(* IEC 61131-3 sources: AXOpen/src/components.drives/ctrl/src/AxoDrives (part 2) *)

            //*************AXO_MOVE_VELOCITY************
            _movementInPositiveDirection := _AxoMoveVelocity_Velocity > 0 AND _AxoMoveVelocity_Direction = AXOpen.Components.Abstractions.Drives.eAxoDriveDirection#PositiveDirection OR
                                            _AxoMoveVelocity_Velocity < 0 AND _AxoMoveVelocity_Direction = AXOpen.Components.Abstractions.Drives.eAxoDriveDirection#NegativeDirection;
            _movementInNegativeDirection := _AxoMoveVelocity_Velocity < 0 AND _AxoMoveVelocity_Direction = AXOpen.Components.Abstractions.Drives.eAxoDriveDirection#PositiveDirection OR
                                            _AxoMoveVelocity_Velocity > 0 AND _AxoMoveVelocity_Direction = AXOpen.Components.Abstractions.Drives.eAxoDriveDirection#NegativeDirection;
                                            AxoMoveVelocity_Task.SetIsDisabled(_movementDisabled OR (_movementInPositiveDirection AND NOT EnablePositive)  OR (_movementInNegativeDirection AND NOT EnableNegative) );
            THIS.MC_MoveVelocity(AxisRef,
                        AxoMoveVelocity_Task.Execute(THIS),
                        _AxoMoveVelocity_ContinuousUpdate,
                        _AxoMoveVelocity_Velocity,
                        _AxoMoveVelocity_Acceleration,
                        _AxoMoveVelocity_Deceleration,
                        _AxoMoveVelocity_Jerk,
                        _AxoMoveVelocity_Direction,
                        AxoMoveVelocity_InVelocity,
                        AxoMoveVelocity_Busy,
                        AxoMoveVelocity_Active,
                        AxoMoveVelocity_CommandAborted,
                        AxoMoveVelocity_Error,
                        AxoMoveVelocity_ErrorID);

            IF AxoMoveVelocity_Task.IsBusy() THEN
                IF AxoMoveVelocity_Task.IsFirstExecutionCycle() THEN
                    AxoMoveVelocity_ContinuousUpdate    :=  _AxoMoveVelocity_ContinuousUpdate;
                    AxoMoveVelocity_Velocity            :=  _AxoMoveVelocity_Velocity;
                    AxoMoveVelocity_Acceleration        :=  _AxoMoveVelocity_Acceleration;
                    AxoMoveVelocity_Deceleration        :=  _AxoMoveVelocity_Deceleration;
                    AxoMoveVelocity_Jerk                :=  _AxoMoveVelocity_Jerk;
                    AxoMoveVelocity_Direction           :=  _AxoMoveVelocity_Direction;
                END_IF;
                AxoMoveVelocity_Task.DoneWhen(AxoMoveVelocity_InVelocity AND NOT _AxoMoveVelocity_ContinuousUpdate);
                AxoMoveVelocity_Task.ThrowWhen(AxoMoveVelocity_Error,CONCAT('<#MC_MoveVelocity has thrown an error: #>', ToString(AxoMoveVelocity_ErrorID)));
                IF AxoMoveVelocity_CommandAborted THEN
                    AxoMoveVelocity_Task.Abort();
                END_IF;
            END_IF;
            IF AxoMoveVelocity_Task.RestoreTriggered() OR AxoMoveVelocity_Task.AbortTriggered() THEN;
                AxoMoveVelocity_InVelocity := FALSE;
            END_IF;
            //******************************************

            //*************AXO_TORQUE_CONTROL***********
            _movementInPositiveDirection := _AxoTorqueControl_Torque > 0 AND _AxoTorqueControl_Direction = AXOpen.Components.Abstractions.Drives.eAxoDriveDirection#PositiveDirection OR
                                            _AxoTorqueControl_Torque < 0 AND _AxoTorqueControl_Direction = AXOpen.Components.Abstractions.Drives.eAxoDriveDirection#NegativeDirection;
            _movementInNegativeDirection := _AxoTorqueControl_Torque < 0 AND _AxoTorqueControl_Direction = AXOpen.Components.Abstractions.Drives.eAxoDriveDirection#PositiveDirection OR
                                            _AxoTorqueControl_Torque > 0 AND _AxoTorqueControl_Direction = AXOpen.Components.Abstractions.Drives.eAxoDriveDirection#NegativeDirection;
            AxoTorqueControl_Task.SetIsDisabled(_movementDisabled OR (_movementInPositiveDirection AND NOT EnablePositive)  OR (_movementInNegativeDirection AND NOT EnableNegative) );
            THIS.MC_TorqueControl(AxisRef,
                        AxoTorqueControl_Task.Execute(THIS),
                        _AxoTorqueControl_ContinuousUpdate,
                        _AxoTorqueControl_Torque,
                        _AxoTorqueControl_TorqueRamp,
                        _AxoTorqueControl_PositionLimit,
                        _AxoTorqueControl_Velocity,
                        _AxoTorqueControl_Acceleration,
                        _AxoTorqueControl_Deceleration,
                        _AxoTorqueControl_Jerk,
                        _AxoTorqueControl_Direction,
                        AxoTorqueControl_InTorque,
                        AxoTorqueControl_Busy,
                        AxoTorqueControl_Active,
                        AxoTorqueControl_CommandAborted,
                        AxoTorqueControl_Error,
                        AxoTorqueControl_ErrorID);

            IF AxoTorqueControl_Task.IsBusy() THEN
                IF AxoTorqueControl_Task.IsFirstExecutionCycle() THEN
                    AxoTorqueControl_ContinuousUpdate   :=  _AxoTorqueControl_ContinuousUpdate;
                    AxoTorqueControl_Torque             :=  _AxoTorqueControl_Torque;
                    AxoTorqueControl_TorqueRamp         :=  _AxoTorqueControl_TorqueRamp;
                    AxoTorqueControl_PositionLimit      :=  _AxoTorqueControl_PositionLimit;
                    AxoTorqueControl_Velocity           :=  _AxoTorqueControl_Velocity;
                    AxoTorqueControl_Acceleration       :=  _AxoTorqueControl_Acceleration;
                    AxoTorqueControl_Deceleration       :=  _AxoTorqueControl_Deceleration;
                    AxoTorqueControl_Jerk               :=  _AxoTorqueControl_Jerk;
                    AxoTorqueControl_Direction          :=  _AxoTorqueControl_Direction;
                END_IF;
                AxoTorqueControl_Task.DoneWhen(AxoTorqueControl_InTorque AND NOT _AxoTorqueControl_ContinuousUpdate);
                AxoTorqueControl_Task.ThrowWhen(AxoTorqueControl_Error,CONCAT('<#MC_TorqueControl has thrown an error: #>', ToString(AxoTorqueControl_ErrorID)));
                IF AxoTorqueControl_CommandAborted THEN
                    AxoTorqueControl_Task.Abort();
                END_IF;
            END_IF;
            IF AxoTorqueControl_Task.RestoreTriggered() OR AxoTorqueControl_Task.AbortTriggered() THEN;
                AxoTorqueControl_InTorque := FALSE;
            END_IF;
            //******************************************
            IF DriveState = eAxoDriveState#ContinuousMotion AND (ActualVelocity > 0.5 AND NOT EnablePositive OR ActualVelocity < -0.5 AND NOT EnableNegative) THEN
                _disabledDuringMovement := TRUE;
                IF AxoMoveVelocity_Task.IsBusy() THEN
                    AxoMoveVelocity_Task.Restore();
                END_IF;
                IF AxoTorqueControl_Task.IsBusy() THEN
                    AxoTorqueControl_Task.Restore();
                END_IF;
            END_IF;
            //*************AXO_SET_POSITION*************
            AxoSetPosition_Task.SetIsDisabled(FALSE);
            THIS.MC_SetPosition(AxisRef,
                        AxoSetPosition_Task.Execute(THIS),
                        _AxoSetPosition_Position,
                        _AxoSetPosition_Relative,
                        _AxoSetPosition_ExecutionMode,
                        AxoSetPosition_Done,
                        AxoSetPosition_Busy,
                        AxoSetPosition_Error,
                        AxoSetPosition_ErrorID);

            IF AxoSetPosition_Task.IsBusy() THEN
                AxoSetPosition_Task.DoneWhen(AxoSetPosition_Done);
                AxoSetPosition_Task.ThrowWhen(AxoSetPosition_Error,CONCAT('<#MC_SetPosition has thrown an error: #>', ToString(AxoSetPosition_ErrorID)));
            END_IF;
            //******************************************

            //*************AXO_SET_OVERRIDE*************
            AxoSetOverride_Task.SetIsDisabled(FALSE);
            AxoSetOverride_Task.Run(THIS);
            THIS.MC_SetOverride(AxisRef,
                        AxoSetOverride_Task.IsSwitchedOn(),
                        _AxoSetOverride_VelFactor,
                        _AxoSetOverride_AccFactor,
                        _AxoSetOverride_JerkFactor,
                        AxoSetOverride_Enabled,
                        AxoSetOverride_Busy,
                        AxoSetOverride_Error,
                        AxoSetOverride_ErrorID);
            //******************************************

            //*************AXO_READ_PARAMETER***********
            AxoReadParameter_Task.SetIsDisabled(FALSE);
            AxoReadParameter_Task.Run(THIS);
            THIS.MC_ReadParameter(AxisRef,
                        AxoReadParameter_Task.IsSwitchedOn(),
                        _AxoReadParameter_ParameterNumber,
                        AxoReadParameter_Valid,
                        AxoReadParameter_Busy,
                        AxoReadParameter_Error,
                        AxoReadParameter_ErrorID,
                        AxoReadParameter_Value);
            IF  AxoReadParameter_Task.IsSwitchedOff() THEN
                AxoReadParameter_Valid := FALSE;
                AxoReadParameter_Value := LINT#0;
            END_IF;
            //******************************************

            //*************AXO_READ_REAL_PARAMETER******
            AxoReadRealParameter_Task.SetIsDisabled(FALSE);
            AxoReadRealParameter_Task.Run(THIS);
            THIS.MC_ReadRealParameter(AxisRef,
                        AxoReadRealParameter_Task.IsSwitchedOn(),
                        _AxoReadRealParameter_ParameterNumber,
                        AxoReadRealParameter_Valid,
                        AxoReadRealParameter_Busy,
                        AxoReadRealParameter_Error,
                        AxoReadRealParameter_ErrorID,
                        AxoReadRealParameter_Value);
            IF  AxoReadRealParameter_Task.IsSwitchedOff() THEN
                AxoReadRealParameter_Valid := FALSE;
                AxoReadRealParameter_Value := REAL#0.0;
            END_IF;
            //******************************************

            //*************AXO_READ_BOOL_PARAMETER******
            AxoReadBoolParameter_Task.SetIsDisabled(FALSE);
            AxoReadBoolParameter_Task.Run(THIS);
            THIS.MC_ReadBoolParameter(AxisRef,
                        AxoReadBoolParameter_Task.IsSwitchedOn(),
                        _AxoReadBoolParameter_ParameterNumber,
                        AxoReadBoolParameter_Valid,
                        AxoReadBoolParameter_Busy,
                        AxoReadBoolParameter_Error,
                        AxoReadBoolParameter_ErrorID,
                        AxoReadBoolParameter_Value);
            IF  AxoReadBoolParameter_Task.IsSwitchedOff() THEN
                AxoReadBoolParameter_Valid := FALSE;
                AxoReadBoolParameter_Value := FALSE;
            END_IF;
            //******************************************

            //*************AXO_WRITE_PARAMETER**********
            AxoWriteParameter_Task.SetIsDisabled(FALSE);
            THIS.MC_WriteParameter(AxisRef,
                        AxoWriteParameter_Task.Execute(THIS),
                        _AxoWriteParameter_ParameterNumber,
                        _AxoWriteParameter_Value,
                        _AxoWriteParameter_ExecutionMode,
                        AxoWriteParameter_Done,
                        AxoWriteParameter_Busy,
                        AxoWriteParameter_Error,
                        AxoWriteParameter_ErrorID);
            IF AxoWriteParameter_Task.IsBusy() THEN
                AxoWriteParameter_Task.DoneWhen(AxoWriteParameter_Done);
                AxoWriteParameter_Task.ThrowWhen(AxoWriteParameter_Error,CONCAT('<#MC_WriteParameter has thrown an error: #>', ToString(AxoWriteParameter_ErrorID)));
            END_IF;
            //******************************************

            //*************AXO_WRITE_REAL_PARAMETER*****
            AxoWriteRealParameter_Task.SetIsDisabled(FALSE);
            THIS.MC_WriteRealParameter(AxisRef,
                        AxoWriteRealParameter_Task.Execute(THIS),
                        _AxoWriteRealParameter_ParameterNumber,
                        _AxoWriteRealParameter_Value,
                        _AxoWriteRealParameter_ExecutionMode,
                        AxoWriteRealParameter_Done,
                        AxoWriteRealParameter_Busy,
                        AxoWriteRealParameter_Error,
                        AxoWriteRealParameter_ErrorID);
            IF AxoWriteRealParameter_Task.IsBusy() THEN
                AxoWriteRealParameter_Task.DoneWhen(AxoWriteRealParameter_Done);
                AxoWriteRealParameter_Task.ThrowWhen(AxoWriteRealParameter_Error,CONCAT('<#MC_WriteRealParameter has thrown an error: #>', ToString(AxoWriteRealParameter_ErrorID)));
            END_IF;
            //******************************************

            //*************AXO_WRITE_BOOL_PARAMETER*****
            AxoWriteBoolParameter_Task.SetIsDisabled(FALSE);
            THIS.MC_WriteBoolParameter(AxisRef,
                        AxoWriteBoolParameter_Task.Execute(THIS),
                        _AxoWriteBoolParameter_ParameterNumber,
                        _AxoWriteBoolParameter_Value,
                        _AxoWriteBoolParameter_ExecutionMode,
                        AxoWriteBoolParameter_Done,
                        AxoWriteBoolParameter_Busy,
                        AxoWriteBoolParameter_Error,
                        AxoWriteBoolParameter_ErrorID);
            IF AxoWriteBoolParameter_Task.IsBusy() THEN
                AxoWriteBoolParameter_Task.DoneWhen(AxoWriteBoolParameter_Done);
                AxoWriteBoolParameter_Task.ThrowWhen(AxoWriteBoolParameter_Error,CONCAT('<#MC_WriteBoolParameter has thrown an error: #>', ToString(AxoWriteBoolParameter_ErrorID)));
            END_IF;
            //******************************************

            //*************AXO_READ_DIGITAL_INPUT*******
            AxoReadDigitalInput_Task.SetIsDisabled(FALSE);
            AxoReadDigitalInput_Task.Run(THIS);
            THIS.MC_ReadDigitalInput(AxisRef,
                        AxoReadDigitalInput_Task.IsSwitchedOn(),
                        _AxoReadDigitalInput_InputNumber,
                        AxoReadDigitalInput_Valid,
                        AxoReadDigitalInput_Busy,
                        AxoReadDigitalInput_Error,
                        AxoReadDigitalInput_ErrorID,
                        AxoReadDigitalInput_Value);
            IF  AxoReadDigitalInput_Task.IsSwitchedOff() THEN
                AxoReadDigitalInput_Valid := FALSE;
                AxoReadDigitalInput_Value := FALSE;
            END_IF;
            //******************************************

            //*************AXO_READ_DIGITAL_OUTPUT******
            AxoReadDigitalOutput_Task.SetIsDisabled(FALSE);
            AxoReadDigitalOutput_Task.Run(THIS);
            THIS.MC_ReadDigitalOutput(AxisRef,
                        AxoReadDigitalOutput_Task.IsSwitchedOn(),
                        _AxoReadDigitalOutput_OutputNumber,
                        AxoReadDigitalOutput_Valid,
                        AxoReadDigitalOutput_Busy,
                        AxoReadDigitalOutput_Error,
                        AxoReadDigitalOutput_ErrorID,
                        AxoReadDigitalOutput_Value);
            IF  AxoReadDigitalOutput_Task.IsSwitchedOff() THEN
                AxoReadDigitalOutput_Valid := FALSE;
                AxoReadDigitalOutput_Value := FALSE;
            END_IF;
            //******************************************

            //*************AXO_WRITE_DIGITAL_OUTPUT*****
            AxoWriteDigitalOutput_Task.SetIsDisabled(FALSE);
            THIS.MC_WriteDigitalOutput(AxisRef,
                        AxoWriteDigitalOutput_Task.Execute(THIS),
                        _AxoWriteDigitalOutput_OutputNumber,
                        _AxoWriteDigitalOutput_Value,
                        _AxoWriteDigitalOutput_ExecutionMode,
                        AxoWriteDigitalOutput_Done,
                        AxoWriteDigitalOutput_Busy,
                        AxoWriteDigitalOutput_Error,
                        AxoWriteDigitalOutput_ErrorID);
            IF AxoWriteDigitalOutput_Task.IsBusy() THEN
                AxoWriteDigitalOutput_Task.DoneWhen(AxoWriteDigitalOutput_Done);
                AxoWriteDigitalOutput_Task.ThrowWhen(AxoWriteDigitalOutput_Error,CONCAT('<#MC_WriteDigitalOutput has thrown an error: #>', ToString(AxoWriteDigitalOutput_ErrorID)));
            END_IF;
            //******************************************

            //*************AXO_READ_ACTUAL_POSITION*****
            AxoReadActualPosition_Task.SetIsDisabled(FALSE);
            AxoReadActualPosition_Task.Run(THIS);
            THIS.MC_ReadActualPosition(AxisRef,
                        AxoReadActualPosition_Task.IsSwitchedOn(),
                        AxoReadActualPosition_Valid,
                        AxoReadActualPosition_Busy,
                        AxoReadActualPosition_Error,
                        AxoReadActualPosition_ErrorID,
                        AxoReadActualPosition_Value);
            IF  AxoReadActualPosition_Task.IsSwitchedOff() THEN
                AxoReadActualPosition_Valid := FALSE;
                AxoReadActualPosition_Value := LREAL#0.0;
            END_IF;
            //******************************************

            //*************AXO_READ_ACTUAL_VELOCITY*****
            AxoReadActualVelocity_Task.SetIsDisabled(FALSE);
            AxoReadActualVelocity_Task.Run(THIS);
            THIS.MC_ReadActualVelocity(AxisRef,
                        AxoReadActualVelocity_Task.IsSwitchedOn(),
                        AxoReadActualVelocity_Valid,
                        AxoReadActualVelocity_Busy,
                        AxoReadActualVelocity_Error,
                        AxoReadActualVelocity_ErrorID,
                        AxoReadActualVelocity_Value);
            IF  AxoReadActualVelocity_Task.IsSwitchedOff() THEN
                AxoReadActualVelocity_Valid := FALSE;
                AxoReadActualVelocity_Value := LREAL#0.0;
            END_IF;
            //******************************************

            //*************AXO_READ_ACTUAL_TORQUE*******
            AxoReadActualTorque_Task.SetIsDisabled(FALSE);
            AxoReadActualTorque_Task.Run(THIS);
            THIS.MC_ReadActualTorque(AxisRef,
                        AxoReadActualTorque_Task.IsSwitchedOn(),
                        AxoReadActualTorque_Valid,
                        AxoReadActualTorque_Busy,
                        AxoReadActualTorque_Error,
                        AxoReadActualTorque_ErrorID,
                        AxoReadActualTorque_Value);
            IF  AxoReadActualTorque_Task.IsSwitchedOff() THEN
                AxoReadActualTorque_Valid := FALSE;
                AxoReadActualTorque_Value := LREAL#0.0;
            END_IF;
            //******************************************

            //*************AXO_READ_STATUS**************
            AxoReadStatus_Task.SetIsDisabled(FALSE);
            AxoReadStatus_Task.Run(THIS);
            THIS.MC_ReadStatus(AxisRef,
                        AxoReadStatus_Task.IsSwitchedOn(),
                        AxoReadStatus_Valid,
                        AxoReadStatus_Busy,
                        AxoReadStatus_Error,
                        AxoReadStatus_ErrorID,
                        AxoReadStatus_ErrorStop,
                        AxoReadStatus_Disabled,
                        AxoReadStatus_Stopping,
                        AxoReadStatus_Homing,
                        AxoReadStatus_Standstill,
                        AxoReadStatus_DiscreteMotion,
                        AxoReadStatus_ContinuousMotion,
                        AxoReadStatus_SynchronizedMotion);
            IF  AxoReadStatus_Task.IsSwitchedOff() THEN
                AxoReadStatus_Valid := FALSE;
                AxoReadStatus_ErrorStop := FALSE;
                AxoReadStatus_Disabled  := FALSE;
                AxoReadStatus_Stopping  := FALSE;
                AxoReadStatus_Homing    := FALSE;
                AxoReadStatus_Standstill    := FALSE;
                AxoReadStatus_DiscreteMotion    := FALSE;
                AxoReadStatus_ContinuousMotion  := FALSE;
                AxoReadStatus_SynchronizedMotion    := FALSE;
            END_IF;
            //******************************************

            //*************AXO_READ_MOTION_STATE********
            AxoReadMotionState_Task.SetIsDisabled(FALSE);
            AxoReadMotionState_Task.Run(THIS);
            THIS.MC_ReadMotionState(AxisRef,
                        AxoReadMotionState_Task.IsSwitchedOn(),
                        _AxoReadMotionState_Source,
                        AxoReadMotionState_Valid,
                        AxoReadMotionState_Busy,
                        AxoReadMotionState_Error,
                        AxoReadMotionState_ErrorID,
                        AxoReadMotionState_ConstantVelocity,
                        AxoReadMotionState_Accelerating,
                        AxoReadMotionState_Decelerating,
                        AxoReadMotionState_DirectionPositive,
                        AxoReadMotionState_DirectionNegative);
            IF  AxoReadMotionState_Task.IsSwitchedOff() THEN
                AxoReadMotionState_Valid := FALSE;
                AxoReadMotionState_ConstantVelocity := FALSE;
                AxoReadMotionState_Accelerating := FALSE;
                AxoReadMotionState_Decelerating := FALSE;
                AxoReadMotionState_DirectionPositive    := FALSE;
                AxoReadMotionState_DirectionNegative    := FALSE;
            END_IF;
            //******************************************

            //*************AXO_READ_AXIS_INFO***********
            AxoReadAxisInfo_Task.SetIsDisabled(FALSE);
            AxoReadAxisInfo_Task.Run(THIS);
            THIS.MC_ReadAxisInfo(AxisRef,
                        AxoReadAxisInfo_Task.IsSwitchedOn(),
                        AxoReadAxisInfo_Valid,
                        AxoReadAxisInfo_Busy,
                        AxoReadAxisInfo_Error,
                        AxoReadAxisInfo_ErrorID,
                        AxoReadAxisInfo_HomeAbsSwitch,
                        AxoReadAxisInfo_LimitSwitchPos,
                        AxoReadAxisInfo_LimitSwitchNeg,
                        AxoReadAxisInfo_Simulation,
                        AxoReadAxisInfo_CommunicationReady,
                        AxoReadAxisInfo_ReadyForPowerOn,
                        AxoReadAxisInfo_PowerOn,
                        AxoReadAxisInfo_IsHomed,
                        AxoReadAxisInfo_AxisWarning);
            IF  AxoReadAxisInfo_Task.IsSwitchedOff() THEN
                AxoReadAxisInfo_Valid := FALSE;
                AxoReadAxisInfo_HomeAbsSwitch   := FALSE;
                AxoReadAxisInfo_LimitSwitchPos  := FALSE;
                AxoReadAxisInfo_LimitSwitchNeg  := FALSE;
                AxoReadAxisInfo_Simulation  := FALSE;
                AxoReadAxisInfo_CommunicationReady  := FALSE;
                AxoReadAxisInfo_ReadyForPowerOn := FALSE;
                AxoReadAxisInfo_PowerOn := FALSE;
                AxoReadAxisInfo_IsHomed := FALSE;
                AxoReadAxisInfo_AxisWarning := FALSE;
            END_IF;
            //******************************************

            //*************AXO_READ_AXIS_ERROR**********
            AxoReadAxisError_Task.SetIsDisabled(FALSE);
            AxoReadAxisError_Task.Run(THIS);
            THIS.MC_ReadAxisError(AxisRef,
                        AxoReadAxisError_Task.IsSwitchedOn(),
                        AxoReadAxisError_Valid,
                        AxoReadAxisError_Busy,
                        AxoReadAxisError_Error,
                        AxoReadAxisError_ErrorID,
                        AxoReadAxisError_AxisErrorID);
            IF  AxoReadAxisError_Task.IsSwitchedOff() THEN
                AxoReadAxisError_Valid := FALSE;
                AxoReadAxisError_ErrorID    := DINT#0;
                AxoReadAxisError_AxisErrorID    := DWORD#0;
            END_IF;
            //******************************************

            //*************AXO_RESET********************
            AxoReset_Task.SetIsDisabled(FALSE);
            THIS.MC_Reset(AxisRef,
                        AxoReset_Task.Execute(THIS),
                        AxoReset_Done,
                        AxoReset_Busy,
                        AxoReset_Error,
                        AxoReset_ErrorID);
            IF AxoReset_Task.IsBusy() THEN
                AxoReset_Task.DoneWhen(AxoReset_Done);
                AxoReset_Task.ThrowWhen(AxoReset_Error,CONCAT('<#MC_Reset has thrown an error: #>', ToString(AxoReset_ErrorID)));
            END_IF;
            //******************************************

            //*************AXO_JOG**********************
            AxoJogPositive.SetIsDisabled(_movementDisabled OR NOT EnablePositive OR AxoJogNegative.IsSwitchedOn());
            AxoJogNegative.SetIsDisabled(_movementDisabled OR NOT EnableNegative OR AxoJogPositive.IsSwitchedOn());
            AxoJogPositive.Run(THIS);
            AxoJogNegative.Run(THIS);
            AxoJogInVelocity                        :=  FALSE;
            AxoJog_Active                           :=  FALSE;
            AxoJog_Done                             :=  FALSE;
            AxoJog_Busy                             :=  FALSE;
            AxoJog_CommandAborted                   :=  FALSE;
            AxoJog_Error                            :=  FALSE;
            AxoJog_ErrorID                          :=  DINT#0;
            IF AxoJogPositive.IsSwitchedOn() THEN
                AxoJog_Direction := AXOpen.Components.Abstractions.Drives.eAxoDriveDirection#PositiveDirection;
            ELSIF AxoJogNegative.IsSwitchedOn() THEN
                AxoJog_Direction := AXOpen.Components.Abstractions.Drives.eAxoDriveDirection#NegativeDirection;
            END_IF;

            IF AxoJogPositive.IsSwitchedOn() AND EnablePositive OR AxoJogNegative.IsSwitchedOn() AND EnableNegative THEN
                IF AxoJogPositive.StartMotion OR AxoJogNegative.StartMotion THEN
                    AxoJogPositive.StartMotion          :=  FALSE;
                    AxoJogNegative.StartMotion          :=  FALSE;
                    AxoHalt_Task.Restore();
                END_IF;
                AxoMoveVelocity_ContinuousUpdate       := FALSE;
                AxoMoveVelocity_Velocity               := AxoJog_Velocity;
                AxoMoveVelocity_Acceleration           := AxoJog_Acceleration;
                AxoMoveVelocity_Deceleration           := AxoJog_Deceleration;
                AxoMoveVelocity_Jerk                   := AxoJog_Jerk;
                AxoMoveVelocity_Direction              := AxoJog_Direction;

                THIS.AxoMoveVelocity();
                AxoJogInVelocity                        :=  AxoMoveVelocity_InVelocity;
                AxoJog_Active                           :=  AxoMoveVelocity_Active;
                AxoJog_Done                             :=  FALSE;
                AxoJog_Busy                             :=  AxoMoveVelocity_Busy;
                AxoJog_CommandAborted                   :=  AxoMoveVelocity_CommandAborted;
                AxoJog_Error                            :=  AxoMoveVelocity_Error;
                AxoJog_ErrorID                          :=  AxoMoveVelocity_ErrorID;
            ELSIF AxoJogPositive.StopMotion OR AxoJogNegative.StopMotion THEN
                AxoMoveVelocity_Task.Restore();
                AxoHalt_Deceleration                   := AxoJog_Deceleration;
                AxoHalt_Jerk                           := AxoJog_Jerk;
                THIS.AxoHalt();
                AxoJogInVelocity                        :=  AxoMoveVelocity_InVelocity;
                AxoJog_Active                           :=  AxoHalt_Active;
                AxoJog_Done                             :=  TRUE;
                AxoJog_Busy                             :=  AxoHalt_Busy;
                AxoJog_CommandAborted                   :=  AxoHalt_CommandAborted;
                AxoJog_Error                            :=  AxoHalt_Error;
                AxoJog_ErrorID                          :=  AxoHalt_ErrorID;
                AxoJogPositive.StopMotion := FALSE;
                AxoJogNegative.StopMotion := FALSE;
            END_IF;
            //******************************************
            ErrorFromMC := FALSE;
            // _warning := FALSE;
            IF AxoPower_Error THEN
                ErrorFromMC := TRUE;
                IF MessageCodeFromMC = ULINT#0 THEN
                    MessageCodeFromMC := TO_ULINT(AxoPower_ErrorID);
                END_IF;
            ELSIF AxoStop_Error THEN
                ErrorFromMC := TRUE;
                IF MessageCodeFromMC = ULINT#0 THEN
                    MessageCodeFromMC := TO_ULINT(AxoStop_ErrorID);
                END_IF;
            ELSIF AxoHalt_Error THEN
                ErrorFromMC := TRUE;
                IF MessageCodeFromMC = ULINT#0 THEN
                    MessageCodeFromMC := TO_ULINT(AxoHalt_ErrorID);
                END_IF;
            ELSIF AxoHome_Error THEN
                ErrorFromMC := TRUE;
                IF MessageCodeFromMC = ULINT#0 THEN
                    MessageCodeFromMC := TO_ULINT(AxoHome_ErrorID);
                END_IF;
            ELSIF AxoMoveAbsolute_Error THEN
                ErrorFromMC := TRUE;
                IF MessageCodeFromMC = ULINT#0 THEN
                    MessageCodeFromMC := TO_ULINT(AxoMoveAbsolute_ErrorID);
                END_IF;
            ELSIF AxoMoveRelative_Error THEN
                ErrorFromMC := TRUE;
                IF MessageCodeFromMC = ULINT#0 THEN
                    MessageCodeFromMC := TO_ULINT(AxoMoveRelative_ErrorID);
                END_IF;
            ELSIF AxoMoveAdditive_Error THEN
                ErrorFromMC := TRUE;
                IF MessageCodeFromMC = ULINT#0 THEN
                    MessageCodeFromMC := TO_ULINT(AxoMoveAdditive_ErrorID);
                END_IF;
            ELSIF AxoMoveVelocity_Error THEN
                ErrorFromMC := TRUE;
                IF MessageCodeFromMC = ULINT#0 THEN
                    MessageCodeFromMC := TO_ULINT(AxoMoveVelocity_ErrorID);
                END_IF;
            ELSIF AxoTorqueControl_Error THEN
                ErrorFromMC := TRUE;
                IF MessageCodeFromMC = ULINT#0 THEN
                    MessageCodeFromMC := TO_ULINT(AxoTorqueControl_ErrorID);
                END_IF;
            ELSIF AxoSetPosition_Error THEN
                ErrorFromMC := TRUE;
                IF MessageCodeFromMC = ULINT#0 THEN
                    MessageCodeFromMC := TO_ULINT(AxoSetPosition_ErrorID);
                END_IF;
            ELSIF AxoSetOverride_Error THEN
                ErrorFromMC := TRUE;
                IF MessageCodeFromMC = ULINT#0 THEN
                    MessageCodeFromMC := TO_ULINT(AxoSetOverride_ErrorID);
                END_IF;
            ELSIF AxoReadParameter_Error THEN
                ErrorFromMC := TRUE;
                IF MessageCodeFromMC = ULINT#0 THEN
                    MessageCodeFromMC := TO_ULINT(AxoReadParameter_ErrorID);
                END_IF;
            ELSIF AxoReadRealParameter_Error THEN
                ErrorFromMC := TRUE;
                IF MessageCodeFromMC = ULINT#0 THEN
                    MessageCodeFromMC := TO_ULINT(AxoReadRealParameter_ErrorID);
                END_IF;
            ELSIF AxoReadBoolParameter_Error THEN
                ErrorFromMC := TRUE;
                IF MessageCodeFromMC = ULINT#0 THEN
                    MessageCodeFromMC := TO_ULINT(AxoReadBoolParameter_ErrorID);
                END_IF;
            ELSIF AxoWriteParameter_Error THEN
                ErrorFromMC := TRUE;
                IF MessageCodeFromMC = ULINT#0 THEN
                    MessageCodeFromMC := TO_ULINT(AxoWriteParameter_ErrorID);
                END_IF;
            ELSIF AxoWriteRealParameter_Error THEN
                ErrorFromMC := TRUE;
                IF MessageCodeFromMC = ULINT#0 THEN
                    MessageCodeFromMC := TO_ULINT(AxoWriteRealParameter_ErrorID);
                END_IF;
            ELSIF AxoWriteBoolParameter_Error THEN
                ErrorFromMC := TRUE;
                IF MessageCodeFromMC = ULINT#0 THEN
                    MessageCodeFromMC := TO_ULINT(AxoWriteBoolParameter_ErrorID);
                END_IF;
            ELSIF AxoReadDigitalInput_Error THEN
                ErrorFromMC := TRUE;
                IF MessageCodeFromMC = ULINT#0 THEN
                    MessageCodeFromMC := TO_ULINT(AxoReadDigitalInput_ErrorID);
                END_IF;
            ELSIF AxoReadDigitalOutput_Error THEN
                ErrorFromMC := TRUE;
                IF MessageCodeFromMC = ULINT#0 THEN
                    MessageCodeFromMC := TO_ULINT(AxoReadDigitalOutput_ErrorID);
                END_IF;
            ELSIF AxoWriteDigitalOutput_Error THEN
                ErrorFromMC := TRUE;
                IF MessageCodeFromMC = ULINT#0 THEN
                    MessageCodeFromMC := TO_ULINT(AxoWriteDigitalOutput_ErrorID);
                END_IF;
            ELSIF AxoReadActualPosition_Error THEN
                ErrorFromMC := TRUE;
                IF MessageCodeFromMC = ULINT#0 THEN
                    MessageCodeFromMC := TO_ULINT(AxoReadActualPosition_ErrorID);
                END_IF;
            ELSIF AxoReadActualVelocity_Error THEN
                ErrorFromMC := TRUE;
                IF MessageCodeFromMC = ULINT#0 THEN
                    MessageCodeFromMC := TO_ULINT(AxoReadActualVelocity_ErrorID);
                END_IF;
            ELSIF AxoReadActualTorque_Error THEN
                ErrorFromMC := TRUE;
                IF MessageCodeFromMC = ULINT#0 THEN
                    MessageCodeFromMC := TO_ULINT(AxoReadActualTorque_ErrorID);
                END_IF;
            ELSIF AxoReadStatus_Error THEN
                ErrorFromMC := TRUE;
                IF MessageCodeFromMC = ULINT#0 THEN
                    MessageCodeFromMC := TO_ULINT(AxoReadStatus_ErrorID);
                END_IF;
            ELSIF AxoReadMotionState_Error THEN
                ErrorFromMC := TRUE;
                IF MessageCodeFromMC = ULINT#0 THEN
                    MessageCodeFromMC := TO_ULINT(AxoReadMotionState_ErrorID);
                END_IF;
            ELSIF AxoReadAxisInfo_Error THEN
                ErrorFromMC := TRUE;
                IF MessageCodeFromMC = ULINT#0 THEN
                    MessageCodeFromMC := TO_ULINT(AxoReadAxisInfo_ErrorID);
                END_IF;
            ELSIF AxoReadAxisError_Error THEN
                ErrorFromMC := TRUE;
                IF MessageCodeFromMC = ULINT#0 THEN
                    MessageCodeFromMC := TO_ULINT(AxoReadAxisError_ErrorID);
                END_IF;
            ELSIF AxoReset_Error THEN
                ErrorFromMC := TRUE;
                IF MessageCodeFromMC = ULINT#0 THEN
                    MessageCodeFromMC := TO_ULINT(AxoReset_ErrorID);
                END_IF;
            ELSIF AxoJog_Error THEN
                ErrorFromMC := TRUE;
                IF MessageCodeFromMC = ULINT#0 THEN
                    MessageCodeFromMC := TO_ULINT(AxoJog_ErrorID);
                END_IF;
            END_IF;

        END_METHOD

        ///<summary>
		/// Restores this instance .
        ///</summary>
        METHOD PUBLIC OVERRIDE Restore
            //AxoPower_Task.Restore();
            AxoStop_Task.Restore();
            AxoHalt_Task.Restore();
            AxoHome_Task.Restore();
            AxoMoveAbsolute_Task.Restore();
            AxoMoveRelative_Task.Restore();
            AxoMoveAdditive_Task.Restore();
            AxoMoveVelocity_Task.Restore();
            AxoTorqueControl_Task.Restore();
            AxoSetPosition_Task.Restore();
            AxoSetOverride_Task.SwitchOff();
            // MC_SetOverride(AxisRef, FALSE);
            AxoReadParameter_Task.SwitchOff();
            // MC_ReadParameter(AxisRef, FALSE);
            AxoReadRealParameter_Task.SwitchOff();
            // MC_ReadRealParameter(AxisRef, FALSE);
            AxoReadBoolParameter_Task.SwitchOff();
            // MC_ReadBoolParameter(AxisRef, FALSE);
            AxoWriteParameter_Task.Restore();
            AxoWriteRealParameter_Task.Restore();
            AxoWriteBoolParameter_Task.Restore();
            AxoReadDigitalInput_Task.SwitchOff();
            // MC_ReadDigitalInput(AxisRef, FALSE);
            AxoReadDigitalOutput_Task.SwitchOff();
            // MC_ReadDigitalOutput(AxisRef, FALSE);
            AxoWriteDigitalOutput_Task.Restore();
            AxoReadActualPosition_Task.SwitchOff();
            // MC_ReadActualPosition(AxisRef, FALSE);
            AxoReadActualVelocity_Task.SwitchOff();
            // MC_ReadActualVelocity(AxisRef, FALSE);
            AxoReadActualTorque_Task.SwitchOff();
            // MC_ReadActualTorque(AxisRef, FALSE);
            AxoReadStatus_Task.SwitchOff();
            // MC_ReadStatus(AxisRef, FALSE);
            AxoReadMotionState_Task.SwitchOff();
            // MC_ReadMotionState(AxisRef, FALSE);
            AxoReadAxisInfo_Task.SwitchOff();
            // MC_ReadAxisInfo(AxisRef, FALSE);
            AxoReadAxisError_Task.SwitchOff();
            // MC_ReadAxisError(AxisRef, FALSE);
            AxoReset_Task.Restore();
            AxoJogPositive.RemoteSwitchOn := FALSE;
            AxoJogPositive.StartMotion := FALSE;
            AxoJogPositive.StopMotion := FALSE;
            AxoJogNegative.RemoteSwitchOn := FALSE;
            AxoJogNegative.StartMotion := FALSE;
            AxoJogNegative.StopMotion := FALSE;

            //************************************************
            MessageCodeFromMC                       :=   ULINT#0;
            ErrorFromMC                             :=   FALSE;
            _movementDisabled                       :=   FALSE;
            _lastMessageCode                        :=   ULINT#0;
            _disabledDuringMovement                 :=   FALSE;
            _movementInPositiveDirection            :=   FALSE;
            _movementInNegativeDirection            :=   FALSE;
            //***********Stop*********************************
            _AxoStop_Deceleration                   :=   LREAL#0.0;
            _AxoStop_Jerk                           :=   LREAL#0.0;
            //***********Halt*********************************
            _AxoHalt_Deceleration                   :=   LREAL#0.0;
            _AxoHalt_Jerk                           :=   LREAL#0.0;
            //***********Home*********************************
            _AxoHome_Position                       :=   LREAL#0.0;
            _AxoHome_HommingMode                    :=   INT#0;
            _AxoHome_Velocity                       :=   LREAL#0.0;
            _AxoHome_Acceleration                   :=   LREAL#0.0;
            _AxoHome_Deceleration                   :=   LREAL#0.0;
            //***********MoveAbsolute*************************
            _AxoMoveAbsolute_ContinuousUpdate       :=   FALSE;
            _AxoMoveAbsolute_Position               :=   LREAL#0.0;
            _AxoMoveAbsolute_Velocity               :=   LREAL#0.0;
            _AxoMoveAbsolute_Acceleration           :=   LREAL#0.0;
            _AxoMoveAbsolute_Deceleration           :=   LREAL#0.0;
            _AxoMoveAbsolute_Jerk                   :=   LREAL#0.0;
            _AxoMoveAbsolute_Direction              :=   AXOpen.Components.Abstractions.Drives.eAxoDriveDirection#CurrentDirection;
            //***********MoveRelative*************************
            _AxoMoveRelative_ContinuousUpdate       :=   FALSE;
            _AxoMoveRelative_Distance               :=   LREAL#0.0;
            _AxoMoveRelative_Velocity               :=   LREAL#0.0;
            _AxoMoveRelative_Acceleration           :=   LREAL#0.0;
            _AxoMoveRelative_Deceleration           :=   LREAL#0.0;
            _AxoMoveRelative_Jerk                   :=   LREAL#0.0;
            //***********MoveAdditive*************************
            _AxoMoveAdditive_ContinuousUpdate       :=   FALSE;
            _AxoMoveAdditive_Distance               :=   LREAL#0.0;
            _AxoMoveAdditive_Velocity               :=   LREAL#0.0;
            _AxoMoveAdditive_Acceleration           :=   LREAL#0.0;
            _AxoMoveAdditive_Deceleration           :=   LREAL#0.0;
            _AxoMoveAdditive_Jerk                   :=   LREAL#0.0;
            //***********MoveVelocity*************************
            _AxoMoveVelocity_ContinuousUpdate       :=   FALSE;
            _AxoMoveVelocity_Velocity               :=   LREAL#0.0;
            _AxoMoveVelocity_Acceleration           :=   LREAL#0.0;
            _AxoMoveVelocity_Deceleration           :=   LREAL#0.0;
            _AxoMoveVelocity_Jerk                   :=   LREAL#0.0;
            _AxoMoveVelocity_Direction              :=   AXOpen.Components.Abstractions.Drives.eAxoDriveDirection#CurrentDirection;
            //***********TorqueControl************************
            _AxoTorqueControl_ContinuousUpdate      :=   FALSE;
            _AxoTorqueControl_Torque                :=   LREAL#0.0;
            _AxoTorqueControl_TorqueRamp            :=   LREAL#0.0;
            _AxoTorqueControl_PositionLimit         :=   LREAL#0.0;
            _AxoTorqueControl_Velocity              :=   LREAL#0.0;
            _AxoTorqueControl_Acceleration          :=   LREAL#0.0;
            _AxoTorqueControl_Deceleration          :=   LREAL#0.0;
            _AxoTorqueControl_Jerk                  :=   LREAL#0.0;
            _AxoTorqueControl_Direction             :=   AXOpen.Components.Abstractions.Drives.eAxoDriveDirection#CurrentDirection;
            //***********SetPosition**************************
            _AxoSetPosition_Position                :=   LREAL#0.0;
            _AxoSetPosition_Relative                :=   FALSE;
            _AxoSetPosition_ExecutionMode           :=   AXOpen.Components.Abstractions.Drives.eAxoExecutionMode#Immediately;
            //***********SetOverride**************************
            _AxoSetOverride_VelFactor               :=   LREAL#0.0;
            _AxoSetOverride_AccFactor               :=   LREAL#0.0;
            _AxoSetOverride_JerkFactor              :=   LREAL#0.0;
            //***********ReadParameter************************
            _AxoReadParameter_ParameterNumber       :=   DINT#0;
            //***********ReadReadParameter************************
            _AxoReadRealParameter_ParameterNumber   :=   DINT#0;
            //***********ReadBoolParameter********************
            _AxoReadBoolParameter_ParameterNumber   :=   DINT#0;
            //***********WriteParameter***********************
            _AxoWriteParameter_ParameterNumber      :=   DINT#0;
            _AxoWriteParameter_Value                :=   LINT#0;
            _AxoWriteParameter_ExecutionMode        :=   AXOpen.Components.Abstractions.Drives.eAxoExecutionMode#Immediately;
            //***********WriteRealParameter***********************
            _AxoWriteRealParameter_ParameterNumber  :=   DINT#0;
            _AxoWriteRealParameter_Value            :=   REAL#0.0;
            _AxoWriteRealParameter_ExecutionMode    :=   AXOpen.Components.Abstractions.Drives.eAxoExecutionMode#Immediately;
            //***********WriteBoolParameter*******************
            _AxoWriteBoolParameter_ParameterNumber  :=   DINT#0;
            _AxoWriteBoolParameter_Value            :=   FALSE;
            _AxoWriteBoolParameter_ExecutionMode    :=   AXOpen.Components.Abstractions.Drives.eAxoExecutionMode#Immediately;
            //***********ReadDigitalInput*********************
            _AxoReadDigitalInput_InputNumber        :=   INT#0;
            //***********ReadDigitalOutput********************
            _AxoReadDigitalOutput_OutputNumber      :=   INT#0;
            //***********WriteDigitalOutput*******************
            _AxoWriteDigitalOutput_OutputNumber     :=   INT#0;
            _AxoWriteDigitalOutput_Value            :=   FALSE;
            _AxoWriteDigitalOutput_ExecutionMode    :=   AXOpen.Components.Abstractions.Drives.eAxoExecutionMode#Immediately;
            //***********ReadMotionState**********************
            _AxoReadMotionState_Source              :=   AXOpen.Components.Abstractions.Drives.eAxoSource#ActualValue;
            //***********Jog**********************************
            _AxoJog_Velocity                        :=   LREAL#0.0;
            _AxoJog_Acceleration                    :=   LREAL#0.0;
            _AxoJog_Deceleration                    :=   LREAL#0.0;
            _AxoJog_Jerk                            :=   LREAL#0.0;
            _AxoJog_Direction                       :=   AXOpen.Components.Abstractions.Drives.eAxoDriveDirection#CurrentDirection;
            _AxoJogInVelocity                       :=   FALSE;
            _AxoJog_Active                          :=   FALSE;
            //************************************************

            RestoreTask.DoneWhen(TRUE);
        END_METHOD

        ///<summary>
		/// Custom logic for the manual control.
        ///</summary>
        METHOD PROTECTED OVERRIDE ManualControl
            //***********Stop*********************************
            _AxoStop_Deceleration                   := AxoStop_Deceleration;
            _AxoStop_Jerk                           := AxoStop_Jerk;
            //***********Halt*********************************
            _AxoHalt_Deceleration                   := AxoHalt_Deceleration;
            _AxoHalt_Jerk                           := AxoHalt_Jerk;
            //***********Home*********************************
            _AxoHome_Position                       := AxoHome_Position;
            _AxoHome_HommingMode                    := AxoHome_HommingMode;
            _AxoHome_Velocity                       := AxoHome_Velocity;
            _AxoHome_Acceleration                   := AxoHome_Acceleration;
            _AxoHome_Deceleration                   := AxoHome_Deceleration;
            //***********MoveAbsolute*************************
            _AxoMoveAbsolute_ContinuousUpdate       := AxoMoveAbsolute_ContinuousUpdate;
            _AxoMoveAbsolute_Position               := AxoMoveAbsolute_Position;
            _AxoMoveAbsolute_Velocity               := AxoMoveAbsolute_Velocity;
            _AxoMoveAbsolute_Acceleration           := AxoMoveAbsolute_Acceleration;
            _AxoMoveAbsolute_Deceleration           := AxoMoveAbsolute_Deceleration;
            _AxoMoveAbsolute_Jerk                   := AxoMoveAbsolute_Jerk;
            _AxoMoveAbsolute_Direction              := AxoMoveAbsolute_Direction;
            //***********MoveRelative*************************
            _AxoMoveRelative_ContinuousUpdate       := AxoMoveRelative_ContinuousUpdate;
            _AxoMoveRelative_Distance               := AxoMoveRelative_Distance;
            _AxoMoveRelative_Velocity               := AxoMoveRelative_Velocity;
            _AxoMoveRelative_Acceleration           := AxoMoveRelative_Acceleration;
            _AxoMoveRelative_Deceleration           := AxoMoveRelative_Deceleration;
            _AxoMoveRelative_Jerk                   := AxoMoveRelative_Jerk;
            //***********MoveAdditive*************************
            _AxoMoveAdditive_ContinuousUpdate       := AxoMoveAdditive_ContinuousUpdate;
            _AxoMoveAdditive_Distance               := AxoMoveAdditive_Distance;
            _AxoMoveAdditive_Velocity               := AxoMoveAdditive_Velocity;
            _AxoMoveAdditive_Acceleration           := AxoMoveAdditive_Acceleration;
            _AxoMoveAdditive_Deceleration           := AxoMoveAdditive_Deceleration;
            _AxoMoveAdditive_Jerk                   := AxoMoveAdditive_Jerk;
            //***********MoveVelocity*************************
            _AxoMoveVelocity_ContinuousUpdate       := AxoMoveVelocity_ContinuousUpdate;
            _AxoMoveVelocity_Velocity               := AxoMoveVelocity_Velocity;
            _AxoMoveVelocity_Acceleration           := AxoMoveVelocity_Acceleration;
            _AxoMoveVelocity_Deceleration           := AxoMoveVelocity_Deceleration;
            _AxoMoveVelocity_Jerk                   := AxoMoveVelocity_Jerk;
            _AxoMoveVelocity_Direction              := AxoMoveVelocity_Direction;
            //***********TorqueControl************************
            _AxoTorqueControl_ContinuousUpdate      := AxoTorqueControl_ContinuousUpdate;
            _AxoTorqueControl_Torque                := AxoTorqueControl_Torque;
            _AxoTorqueControl_TorqueRamp            := AxoTorqueControl_TorqueRamp;
            _AxoTorqueControl_PositionLimit         := AxoTorqueControl_PositionLimit;
            _AxoTorqueControl_Velocity              := AxoTorqueControl_Velocity;
            _AxoTorqueControl_Acceleration          := AxoTorqueControl_Acceleration;
            _AxoTorqueControl_Deceleration          := AxoTorqueControl_Deceleration;
            _AxoTorqueControl_Jerk                  := AxoTorqueControl_Jerk;
            _AxoTorqueControl_Direction             := AxoTorqueControl_Direction;
            //***********SetPosition**************************
            _AxoSetPosition_Position                := AxoSetPosition_Position;
            _AxoSetPosition_Relative                := AxoSetPosition_Relative;
            _AxoSetPosition_ExecutionMode           := AxoSetPosition_ExecutionMode;
            //***********SetOverride**************************
            _AxoSetOverride_VelFactor               := AxoSetOverride_VelFactor;
            _AxoSetOverride_AccFactor               := AxoSetOverride_AccFactor;
            _AxoSetOverride_JerkFactor              := AxoSetOverride_JerkFactor;
            //***********ReadParameter************************
            _AxoReadParameter_ParameterNumber       := AxoReadParameter_ParameterNumber;
            //***********ReadRealParameter************************
            _AxoReadRealParameter_ParameterNumber       := AxoReadRealParameter_ParameterNumber;
            //***********ReadBoolParameter********************
            _AxoReadBoolParameter_ParameterNumber   := AxoReadBoolParameter_ParameterNumber;
            //***********WriteParameter***********************
            _AxoWriteParameter_ParameterNumber      := AxoWriteParameter_ParameterNumber;
            _AxoWriteParameter_Value                := AxoWriteParameter_Value;
            _AxoWriteParameter_ExecutionMode        := AxoWriteParameter_ExecutionMode;
            //***********WriteRealParameter*******************
            _AxoWriteRealParameter_ParameterNumber  := AxoWriteRealParameter_ParameterNumber;
            _AxoWriteRealParameter_Value            := AxoWriteRealParameter_Value;
            _AxoWriteRealParameter_ExecutionMode    := AxoWriteRealParameter_ExecutionMode;
            //***********WriteBoolParameter*******************
            _AxoWriteBoolParameter_ParameterNumber  := AxoWriteBoolParameter_ParameterNumber;
            _AxoWriteBoolParameter_Value            := AxoWriteBoolParameter_Value;
            _AxoWriteBoolParameter_ExecutionMode    := AxoWriteBoolParameter_ExecutionMode;
            //***********ReadDigitalInput*********************
            _AxoReadDigitalInput_InputNumber        := AxoReadDigitalInput_InputNumber;
            //***********ReadDigitalOutput********************
            _AxoReadDigitalOutput_OutputNumber      := AxoReadDigitalOutput_OutputNumber;
            //***********WriteDigitalOutput*******************
            _AxoWriteDigitalOutput_OutputNumber     := AxoWriteDigitalOutput_OutputNumber;
            _AxoWriteDigitalOutput_Value            := AxoWriteDigitalOutput_Value;
            _AxoWriteDigitalOutput_ExecutionMode    := AxoWriteDigitalOutput_ExecutionMode;
            //***********ReadMotionState**********************
            _AxoReadMotionState_Source              := AxoReadMotionState_Source;
            //***********Jog**********************************
            _AxoJog_Velocity                        := AxoJog_Velocity;
            _AxoJog_Acceleration                    := AxoJog_Acceleration;
            _AxoJog_Deceleration                    := AxoJog_Deceleration;
            _AxoJog_Jerk                            := AxoJog_Jerk;
            _AxoJog_Direction                       := AxoJog_Direction;
            _AxoJogInVelocity                       := AxoJogInVelocity;
            _AxoJog_Active                          := AxoJog_Active;

            IF AxoJog_Active THEN
                _AxoMoveVelocity_ContinuousUpdate       := FALSE;
                _AxoMoveVelocity_Velocity               := AxoJog_Velocity;
                _AxoMoveVelocity_Acceleration           := AxoJog_Acceleration;
                _AxoMoveVelocity_Deceleration           := AxoJog_Deceleration;
                _AxoMoveVelocity_Jerk                   := AxoJog_Jerk;
                _AxoMoveVelocity_Direction              := AxoJog_Direction;

                _AxoHalt_Deceleration                   := AxoJog_Deceleration;
                _AxoHalt_Jerk                           := AxoJog_Jerk;
            END_IF;
            //************************************************
            AxoPower_Task.Manual();
        END_METHOD

        ///<summary>
        /// This method commands the axis to perform the «search home» sequence. The ‘Position’ input is used to set the absolute
        /// position when reference signal is detected. This method completes at ‘Standstill’ if it was started in ‘Standstill’.
        ///</summary>
        METHOD PUBLIC AxoHome   : IAxoTaskState
            VAR_INPUT
                Position        :   LREAL;                      //  Absolute position when the reference signal is detected
                HommingMode     :   INT;                        //  Required homming mode
                Velocity        :   LREAL;                      //  Value of the maximum ‘Velocity’ (not necessarily reached) [u/s].
                Acceleration    :   LREAL;                      //  Value of the ‘Acceleration’ (always positive) (increasing energy of the motor) [u/s2]
                Deceleration    :   LREAL;                      //  Value of the ‘Deceleration’ (always positive) (decreasing energy of the motor) [u/s2]
            END_VAR
            VAR_OUTPUT
                Done            :   BOOL;                       // Reference known and set sucessfully
                Busy            :   BOOL;                       // The method is not finished and new output values are to be expected
                Active          :   BOOL;                       // Indicates that the method has control on the axis
                CommandAborted  :   BOOL;                       // ‘Command’ is aborted by another command
                Error           :   BOOL;                       // Signals that an error has occurred within the method
                ErrorID         :   DINT;                       // Error identification
             END_VAR

            _AxoHome_Position    :=  Position;
            _AxoHome_HommingMode :=  HommingMode;
            _AxoHome_Velocity    :=  Velocity;
            _AxoHome_Acceleration:=  Acceleration;
            _AxoHome_Deceleration:=  Deceleration;

            Done            :=  AxoHome_Done;
            Busy            :=  AxoHome_Busy;
            Active          :=  AxoHome_Active;
            CommandAborted  :=  AxoHome_CommandAborted;
            Error           :=  AxoHome_Error;
            ErrorID         :=  AxoHome_ErrorID;

            AxoHome := AxoHome_Task.Invoke(THIS);
        END_METHOD

        ///<summary>
        /// This method commands a controlled motion stop and transfers the axis to the state ‘Stopping’. It aborts any
        /// ongoing method execution. While the axis is in state ‘Stopping’, no other method can perform any motion on this axis.
        ///</summary>
        METHOD PUBLIC AxoStop   : IAxoTaskState
            VAR_INPUT
                Deceleration    :   LREAL;                      //  Value of the ‘Deceleration’ [u/s2]
                Jerk            :   LREAL;                      //  Value of the ‘Jerk’ [u/s3]
            END_VAR
            VAR_OUTPUT
                Done            :   BOOL;                       // Zero velocity reached
                Busy            :   BOOL;                       // The method is not finished and new output values are to be expected
                Active          :   BOOL;                       // Indicates that the method has control on the axis
                CommandAborted  :   BOOL;                       // ‘Command’ is aborted by switching off power (only possibility to abort)
                Error           :   BOOL;                       // Signals that an error has occurred within the method
                ErrorID         :   DINT;                       // Error identification
             END_VAR

            _AxoStop_Deceleration   :=  Deceleration;
            _AxoStop_Jerk           :=  Jerk;

            Done            :=  AxoStop_Done;
            Busy            :=  AxoStop_Busy;
            Active          :=  AxoStop_Active;
            CommandAborted  :=  AxoStop_CommandAborted;
            Error           :=  AxoStop_Error;
            ErrorID         :=  AxoStop_ErrorID;

            AxoStop := AxoStop_Task.Invoke(THIS);
        END_METHOD

        ///<summary>
        /// This method commands a controlled motion stop. The axis is moved to the state ‘DiscreteMotion’, until the
        /// velocity is zero. With the ‘Done’ output set, the state is transferred to ‘Standstill’.
        ///</summary>
        METHOD PUBLIC AxoHalt : IAxoTaskState
            VAR_INPUT
                Deceleration    :   LREAL;                      //  Value of the ‘Deceleration’ [u/s2]
                Jerk            :   LREAL;                      //  Value of the ‘Jerk’ [u/s3]
            END_VAR
            VAR_OUTPUT
                Done            :   BOOL;                       // Zero velocity reached
                Busy            :   BOOL;                       // The method is not finished and new output values are to be expected
                Active          :   BOOL;                       // Indicates that the method has control on the axis
                CommandAborted  :   BOOL;                       // ‘Command’ is aborted by switching off power (only possibility to abort)
                Error           :   BOOL;                       // Signals that an error has occurred within the method
                ErrorID         :   DINT;                       // Error identification
             END_VAR

            _AxoHalt_Deceleration   :=  Deceleration;
            _AxoHalt_Jerk           :=  Jerk;

            Done            :=  AxoHalt_Done;
            Busy            :=  AxoHalt_Busy;
            Active          :=  AxoHalt_Active;
            CommandAborted  :=  AxoHalt_CommandAborted;
            Error           :=  AxoHalt_Error;
            ErrorID         :=  AxoHalt_ErrorID;

            AxoHalt := AxoHalt_Task.Invoke(THIS);
        END_METHOD

        ///<summary>
        /// This method commands a controlled motion to a specified absolute position.
        ///<summary>
        METHOD PUBLIC AxoMoveAbsolute : IAxoTaskState
            VAR_INPUT
                ContinuousUpdate:   BOOL;                       //  Activate ‘ContinuousUpdate’ - target parameters should be changed during movement
                Position        :   LREAL;                      //  Commanded ‘Position’ for the motion (in technical unit [u]) (negative or positive)
                Velocity        :   LREAL;                      //  Value of the maximum ‘Velocity’ (not necessarily reached) [u/s].
                Acceleration    :   LREAL;                      //  Value of the ‘Acceleration’ (always positive) (increasing energy of the motor) [u/s2]
                Deceleration    :   LREAL;                      //  Value of the ‘Deceleration’ (always positive) (decreasing energy of the motor) [u/s2]
                Jerk            :   LREAL;                      //  Value of the ‘Jerk’ [u/s3]
                Direction       :   AXOpen.Components.Abstractions.Drives.eAxoDriveDirection;         //  Enum type (1-of-4 values: PositiveDirection, ShortestWay, NegativeDirection, CurrentDirection)
            END_VAR
            VAR_OUTPUT
                Done            :   BOOL;                       // Commanded position finally reached
                Busy            :   BOOL;                       // The method is not finished and new output values are to be expected
                Active          :   BOOL;                       // Indicates that the method has control on the axis
                CommandAborted  :   BOOL;                       // ‘Command’ is aborted by another command
                Error           :   BOOL;                       // Signals that an error has occurred within the method
                ErrorID         :   DINT;                       // Error identification
             END_VAR

            _AxoMoveAbsolute_ContinuousUpdate   := ContinuousUpdate;
            _AxoMoveAbsolute_Position           := Position;
            _AxoMoveAbsolute_Velocity           := Velocity;
            _AxoMoveAbsolute_Acceleration       := Acceleration;
            _AxoMoveAbsolute_Deceleration       := Deceleration;
            _AxoMoveAbsolute_Jerk               := Jerk;
            _AxoMoveAbsolute_Direction          := Direction;

            Done            :=  AxoMoveAbsolute_Done;
            Busy            :=  AxoMoveAbsolute_Busy;
            Active          :=  AxoMoveAbsolute_Active;
            CommandAborted  :=  AxoMoveAbsolute_CommandAborted;
            Error           :=  AxoMoveAbsolute_Error;
            ErrorID         :=  AxoMoveAbsolute_ErrorID;

            AxoMoveAbsolute := AxoMoveAbsolute_Task.Invoke(THIS);
        END_METHOD

        ///<summary>
        /// This method  commands a controlled motion of a specified distance relative to the set position at the time of the execution.
        ///<summary>
        METHOD PUBLIC AxoMoveRelative : IAxoTaskState
            VAR_INPUT
                ContinuousUpdate:   BOOL;                       //  Activate ‘ContinuousUpdate’ - target parameters should be changed during movement
                Distance        :   LREAL;                      //  Relative distance for the motion (in technical unit [u]
                Velocity        :   LREAL;                      //  Value of the maximum ‘Velocity’ (not necessarily reached) [u/s].
                Acceleration    :   LREAL;                      //  Value of the ‘Acceleration’ (always positive) (increasing energy of the motor) [u/s2]
                Deceleration    :   LREAL;                      //  Value of the ‘Deceleration’ (always positive) (decreasing energy of the motor) [u/s2]
                Jerk            :   LREAL;                      //  Value of the ‘Jerk’ [u/s3]
            END_VAR
            VAR_OUTPUT
                Done            :   BOOL;                       // Commanded distance reached
                Busy            :   BOOL;                       // The method is not finished and new output values are to be expected
                Active          :   BOOL;                       // Indicates that the method has control on the axis
                CommandAborted  :   BOOL;                       // ‘Command’ is aborted by another command
                Error           :   BOOL;                       // Signals that an error has occurred within the method
                ErrorID         :   DINT;                       // Error identification
             END_VAR

            _AxoMoveRelative_ContinuousUpdate   :=  ContinuousUpdate;
            _AxoMoveRelative_Distance           :=  Distance;
            _AxoMoveRelative_Velocity           :=  Velocity;
            _AxoMoveRelative_Acceleration       :=  Acceleration;
            _AxoMoveRelative_Deceleration       :=  Deceleration;
            _AxoMoveRelative_Jerk               :=  Jerk;

            Done            :=  AxoMoveRelative_Done;
            Busy            :=  AxoMoveRelative_Busy;
            Active          :=  AxoMoveRelative_Active;
            CommandAborted  :=  AxoMoveRelative_CommandAborted;
            Error           :=  AxoMoveRelative_Error;
            ErrorID         :=  AxoMoveRelative_ErrorID;

            AxoMoveRelative :=  AxoMoveRelative_Task.Invoke(THIS);
        END_METHOD

        ///<summary>
        /// This method commands a controlled motion of a specified relative distance additional to the most recent
        /// commanded position in the axis state ‘DiscreteMotion’. The most recent commanded position may be the result of a
        /// previous MC_MoveAdditive motion which was aborted. If the method is activated in the axis state ‘ContinuousMotion’, the
        /// specified relative distance is added to the set position at the time of the execution.
        ///<summary>
        METHOD PUBLIC AxoMoveAdditive  : IAxoTaskState
            VAR_INPUT
                ContinuousUpdate:   BOOL;                       //  Activate ‘ContinuousUpdate’ - target parameters should be changed during movement
                Distance        :   LREAL;                      //  Relative distance for the motion (in technical unit [u]
                Velocity        :   LREAL;                      //  Value of the maximum ‘Velocity’ (not necessarily reached) [u/s].
                Acceleration    :   LREAL;                      //  Value of the ‘Acceleration’ (always positive) (increasing energy of the motor) [u/s2]
                Deceleration    :   LREAL;                      //  Value of the ‘Deceleration’ (always positive) (decreasing energy of the motor) [u/s2]
                Jerk            :   LREAL;                      //  Value of the ‘Jerk’ [u/s3]
            END_VAR
            VAR_OUTPUT
                Done            :   BOOL;                       // Commanded distance reached
                Busy            :   BOOL;                       // The method is not finished and new output values are to be expected
                Active          :   BOOL;                       // Indicates that the method has control on the axis
                CommandAborted  :   BOOL;                       // ‘Command’ is aborted by another command
                Error           :   BOOL;                       // Signals that an error has occurred within the method
                ErrorID         :   DINT;                       // Error identification
             END_VAR

            _AxoMoveAdditive_ContinuousUpdate   :=  ContinuousUpdate;
            _AxoMoveAdditive_Distance           :=  Distance;
            _AxoMoveAdditive_Velocity           :=  Velocity;
            _AxoMoveAdditive_Acceleration       :=  Acceleration;
            _AxoMoveAdditive_Deceleration       :=  Deceleration;
            _AxoMoveAdditive_Jerk               :=  Jerk;

            Done            :=  AxoMoveAdditive_Done;
            Busy            :=  AxoMoveAdditive_Busy;
            Active          :=  AxoMoveAdditive_Active;
            CommandAborted  :=  AxoMoveAdditive_CommandAborted;
            Error           :=  AxoMoveAdditive_Error;
            ErrorID         :=  AxoMoveAdditive_ErrorID;

            AxoMoveAdditive := AxoMoveAdditive_Task.Invoke(THIS);
        END_METHOD

        ///<summary>
        /// This method commands a never ending controlled motion at a specified velocity.
        ///<summary>
        METHOD PUBLIC AxoMoveVelocity  : IAxoTaskState
            VAR_INPUT
                ContinuousUpdate:   BOOL;                       //  Activate ‘ContinuousUpdate’ - target parameters should be changed during movement
                Velocity        :   LREAL;                      //  Value of the maximum velocity [u/s]. Can be a signed value.
                Acceleration    :   LREAL;                      //  Value of the ‘Acceleration’ (always positive) (increasing energy of the motor) [u/s2]
                Deceleration    :   LREAL;                      //  Value of the ‘Deceleration’ (always positive) (decreasing energy of the motor) [u/s2]
                Jerk            :   LREAL;                      //  Value of the ‘Jerk’ [u/s3]
                Direction       :   AXOpen.Components.Abstractions.Drives.eAxoDriveDirection;         //  Enum type (1-of-3 values: PositiveDirection, NegativeDirection, and CurrentDirection. Note: shortest way not applicable)
            END_VAR
            VAR_OUTPUT
                InVelocity      :   BOOL;                       // Commanded velocity reached
                Busy            :   BOOL;                       // The method is not finished and new output values are to be expected
                Active          :   BOOL;                       // Indicates that the method has control on the axis
                CommandAborted  :   BOOL;                       // ‘Command’ is aborted by another command
                Error           :   BOOL;                       // Signals that an error has occurred within the method
                ErrorID         :   DINT;                       // Error identification
             END_VAR

            _AxoMoveVelocity_ContinuousUpdate   :=  ContinuousUpdate;
            _AxoMoveVelocity_Velocity           :=  Velocity;
            _AxoMoveVelocity_Acceleration       :=  Acceleration;
            _AxoMoveVelocity_Deceleration       :=  Deceleration;
            _AxoMoveVelocity_Jerk               :=  Jerk;
            _AxoMoveVelocity_Direction          :=  Direction;

            InVelocity      :=  AxoMoveVelocity_InVelocity;
            Busy            :=  AxoMoveVelocity_Busy;
            Active          :=  AxoMoveVelocity_Active;
            CommandAborted  :=  AxoMoveVelocity_CommandAborted;
            Error           :=  AxoMoveVelocity_Error;
            ErrorID         :=  AxoMoveVelocity_ErrorID;

            AxoMoveVelocity := AxoMoveVelocity_Task.Invoke(THIS);
        END_METHOD

        ///<summary>
        /// This method continuously exerts a torque or force of the specified magnitude. This magnitude is
        /// approached using a defined ramp (‘TorqueRamp’), and the method sets the ‘InTorque’ output if the
        /// commanded torque level is reached. This method is applicable for force and torque. When there is no external
        /// load, force is applicable. Positive torque is in the positive direction of velocity.
        ///<summary>
        METHOD PUBLIC AxoTorqueControl : IAxoTaskState
            VAR_INPUT
                ContinuousUpdate:   BOOL;                       //  Activate ‘ContinuousUpdate’ - target parameters should be changed during movement
                Torque          :   LREAL;                      //  Value of the torque (Torque or force in technical unit [u])
                TorqueRamp      :   LREAL;                      //  The maximum time derivative of the set value of the torque or force (in technical unit per sec. [u/s])
                PositionLimit   :   LREAL;                      //  Position limit.
                Velocity        :   LREAL;                      //  Absolute value of the maximum velocity.
                Acceleration    :   LREAL;                      //  Value of the maximum acceleration (acceleration is applicable with same sign of torque and velocity)
                Deceleration    :   LREAL;                      //  Value of the maximum deceleration (deceleration is applicable with opposite signs of torque and velocity)
                Jerk            :   LREAL;                      //  Value of the maximum jerk
                Direction       :   AXOpen.Components.Abstractions.Drives.eAxoDriveDirection;         //  Enum type (1 of 2 values: PositiveDirection, NegativeDirection or CurrentDirection). Specifies the direction of the torque. (Note: Torque input can be signed value).
            END_VAR
            VAR_OUTPUT
                InTorque        :   BOOL;                       //  Setpoint value of torque or force equals the commandedvalue
                Busy            :   BOOL;                       //  The method is not finished and new output values are to be expected
                Active          :   BOOL;                       //  Indicates that the method has control on the axis
                CommandAborted  :   BOOL;                       //  ‘Command’ is aborted by another command
                Error           :   BOOL;                       //  Signals that an error has occurred within the method
                ErrorID         :   DINT;                       //  Error identification
            END_VAR

            _AxoTorqueControl_ContinuousUpdate  :=  ContinuousUpdate;
            _AxoTorqueControl_Torque            :=  Torque;
            _AxoTorqueControl_TorqueRamp        :=  TorqueRamp;
            _AxoTorqueControl_PositionLimit     :=  PositionLimit;
            _AxoTorqueControl_Velocity          :=  Velocity;
            _AxoTorqueControl_Acceleration      :=  Acceleration;
            _AxoTorqueControl_Deceleration      :=  Deceleration;
            _AxoTorqueControl_Jerk              :=  Jerk;
            _AxoTorqueControl_Direction         :=  Direction;

            InTorque        :=  AxoTorqueControl_InTorque;
            Busy            :=  AxoTorqueControl_Busy;
            Active          :=  AxoTorqueControl_Active;
            CommandAborted  :=  AxoTorqueControl_CommandAborted;
            Error           :=  AxoTorqueControl_Error;
            ErrorID         :=  AxoTorqueControl_ErrorID;

            AxoTorqueControl    := AxoTorqueControl_Task.Invoke(THIS);
        END_METHOD

        ///<summary>
        /// This method shifts the coordinate system of an axis by manipulating both the set-point position as well as the
        /// actual position of an axis with the same value without any movement caused. (Re-calibration with same following error).
        /// This can be used for instance for a reference situation. This method can also be used during motion without changing
        /// the commanded position, which is now positioned in the shifted coordinate system.
        ///<summary>
        METHOD PUBLIC AxoSetPosition   : IAxoTaskState
            VAR_INPUT
                Position        :   LREAL;                      //  Position unit [u] (Means ‘Distance’ if ‘Relative’= TRUE)
                Relative        :   BOOL;                       //  ‘Relative’ distance if True, ‘Absolute’ position if False (= Default)
                ExecutionMode   :   AXOpen.Components.Abstractions.Drives.eAxoExecutionMode;          //  Defines the chronological sequence of the method.
            END_VAR
            VAR_OUTPUT
                Done            :   BOOL;                       //  ‘Position’ has new value
                Error           :   BOOL;                       //  Signals that an error has occurred within the FunctionBlock
                ErrorID         :   DINT;                       //  Error identification
            END_VAR

            _AxoSetPosition_Position         :=  Position;
            _AxoSetPosition_Relative         :=  Relative;
            _AxoSetPosition_ExecutionMode    :=  ExecutionMode;

            Done            :=  AxoSetPosition_Done;
            Error           :=  AxoSetPosition_Error;
            ErrorID         :=  AxoSetPosition_ErrorID;

            AxoSetPosition := AxoSetPosition_Task.Invoke(THIS);
        END_METHOD

        ///<summary>
        /// This method sets the values of override for the whole axis, and all functions that are working on that axis. The override
        /// parameters contribute as a factor to the calculation of the commanded velocity, acceleration and jerk of the motion.
        ///<summary>
        METHOD PUBLIC AxoSetOverride   : IAxoToggleTask
            VAR_INPUT
                Enable          :   BOOL;                       //  If SET, it writes the value of the override factor continuously. If RESET it should keep the last value.
                VelFactor       :   LREAL;                      //  New override factor for the velocity
                AccFactor       :   LREAL;                      //  New override factor for the acceleration/deceleration
                JerkFactor      :   LREAL;                      //  New override factor for the jer
            END_VAR
            VAR_OUTPUT
                Enabled         :   BOOL;                       //  Signals that the override factor(s) is (are) set successfully
                Busy            :   BOOL;                       //  The method is not finished and new output values are to be expected
                Error           :   BOOL;                       //  Signals that an error has occurred within the FumethodnctionBlock
                ErrorID         :   DINT;                       //  Error identification
            END_VAR

            IF Enable THEN
                _AxoSetOverride_VelFactor   :=  VelFactor;
                _AxoSetOverride_AccFactor   :=  AccFactor;
                _AxoSetOverride_JerkFactor  :=  JerkFactor;

                AxoSetOverride_Task.SwitchOn();
            ELSE
                AxoSetOverride_Task.SwitchOff();
                // THIS.MC_SetOverride(AxisRef, FALSE);
            END_IF;

            AxoSetOverride  := AxoSetOverride_Task;
        END_METHOD

        ///<summary>
        /// This method returns the value of a vendor specific parameter. The returned Value has to be converted to Real
        /// if necessary. If not possible, the vendor has to supply a vendor specific method to read the parameter.
        ///<summary>
        METHOD PUBLIC AxoReadParameter : IAxoToggleTask
            VAR_INPUT
                Enable          :   BOOL;                       //  Get the value of the parameter continuously while enabled
                ParameterNumber :   DINT;                       //  Number of the parameter. One can also use symbolic parameter names which are declared as VAR CONST.
            END_VAR
            VAR_OUTPUT
                Valid           :   BOOL;                       //  A valid output is available at the method
                Busy            :   BOOL;                       //  The method is not finished and new output values are to be expected
                Error           :   BOOL;                       //  Signals that an error has occurred within the method
                ErrorID         :   DINT;                       //  Error identification
                Value           :   LINT;                       //  Value of the specified parameter in the datatype, as specified by the vendor
            END_VAR

            IF Enable THEN
                _AxoReadParameter_ParameterNumber   :=  ParameterNumber;

                AxoReadParameter_Task.SwitchOn();
            ELSE
                AxoReadParameter_Task.SwitchOff();
                // THIS.MC_ReadParameter(AxisRef, FALSE);
            END_IF;

            Valid   := AxoReadParameter_Valid;
            Busy    := AxoReadParameter_Busy;
            Error   := AxoReadParameter_Error;
            ErrorID := AxoReadParameter_ErrorID;
            Value   := AxoReadParameter_Value;

            AxoReadParameter  := AxoReadParameter_Task;
        END_METHOD

        ///<summary>
        /// This method returns the value of a vendor specific parameter with datatype REAL
        ///<summary>
        METHOD PUBLIC AxoReadRealParameter : IAxoToggleTask
            VAR_INPUT
                Enable          :   BOOL;                       //  Get the value of the parameter continuously while enabled
                ParameterNumber :   DINT;                       //  Number of the parameter. One can also use symbolic parameter names which are declared as VAR CONST.
            END_VAR
            VAR_OUTPUT
                Valid           :   BOOL;                       //  A valid output is available at the method
                Busy            :   BOOL;                       //  The method is not finished and new output values are to be expected
                Error           :   BOOL;                       //  Signals that an error has occurred within the method
                ErrorID         :   DINT;                       //  Error identification
                Value           :   REAL;                       //  Value of the specified parameter in the datatype, as specified by the vendor
            END_VAR

            IF Enable THEN
                _AxoReadRealParameter_ParameterNumber   :=  ParameterNumber;

                AxoReadRealParameter_Task.SwitchOn();
            ELSE
                AxoReadRealParameter_Task.SwitchOff();
                // THIS.MC_ReadRealParameter(AxisRef, FALSE);
            END_IF;

            Valid   := AxoReadRealParameter_Valid;
            Busy    := AxoReadRealParameter_Busy;
            Error   := AxoReadRealParameter_Error;
            ErrorID := AxoReadRealParameter_ErrorID;
            Value   := AxoReadRealParameter_Value;

            AxoReadRealParameter  := AxoReadRealParameter_Task;
        END_METHOD

        ///<summary>
        /// This method returns the value of a vendor specific parameter with datatype BOOL.
        ///<summary>
        METHOD PUBLIC AxoReadBoolParameter : IAxoToggleTask
            VAR_INPUT
                Enable          :   BOOL;                       //  Get the value of the parameter continuously while enabled
                ParameterNumber :   DINT;                       //  Number of the parameter. One can also use symbolic parameter names which are declared as VAR CONST.
            END_VAR
            VAR_OUTPUT
                Valid           :   BOOL;                       //  A valid output is available at the method
                Busy            :   BOOL;                       //  The method is not finished and new output values are to be expected
                Error           :   BOOL;                       //  Signals that an error has occurred within the method
                ErrorID         :   DINT;                       //  Error identification
                Value           :   BOOL;                       //  Value of the specified parameter in the datatype, as specified by the vendor
            END_VAR

            IF Enable THEN
                _AxoReadBoolParameter_ParameterNumber   :=  ParameterNumber;

                AxoReadBoolParameter_Task.SwitchOn();
            ELSE
                AxoReadBoolParameter_Task.SwitchOff();
                // THIS.MC_ReadBoolParameter(AxisRef, FALSE);
            END_IF;

            Valid   := AxoReadBoolParameter_Valid;
            Busy    := AxoReadBoolParameter_Busy;
            Error   := AxoReadBoolParameter_Error;
            ErrorID := AxoReadBoolParameter_ErrorID;
            Value   := AxoReadBoolParameter_Value;

            AxoReadBoolParameter  := AxoReadBoolParameter_Task;
        END_METHOD

        ///<summary>
        /// This method modifies the value of a vendor specific parameter.
        ///<summary>
        METHOD PUBLIC AxoWriteParameter : IAxoTaskState
            VAR_INPUT
                ParameterNumber :   DINT;                       //  Number of the parameter (correspondence between number andparameter is specified in the table above)
                Value           :   LINT;                       //  New value of the specified parameter
                ExecutionMode   :   AXOpen.Components.Abstractions.Drives.eAxoExecutionMode;          //  Defines the chronological sequence of the method.
            END_VAR
            VAR_OUTPUT
                Done            :   BOOL;                       //  Parameter successfully written
                Busy            :   BOOL;                       //  The method is not finished and new output values are to be expected.
                Error           :   BOOL;                       //  Signals that an error has occurred within the method
                ErrorID         :   DINT;                       //  Error identification
            END_VAR

            _AxoWriteParameter_ParameterNumber  :=  ParameterNumber;
            _AxoWriteParameter_Value            :=  Value;
            _AxoWriteParameter_ExecutionMode    :=  ExecutionMode;

            Done                :=  AxoWriteParameter_Done;
            Busy                :=  AxoWriteParameter_Busy;
            Error               :=  AxoWriteParameter_Error;
            ErrorID             :=  AxoWriteParameter_ErrorID;

            AxoWriteParameter   :=  AxoWriteParameter_Task.Invoke(THIS);
        END_METHOD

        ///<summary>
        /// This method modifies the value of a vendor specific parameter of type REAL.
        ///<summary>
        METHOD PUBLIC AxoWriteRealParameter    : IAxoTaskState
            VAR_INPUT
                ParameterNumber :   DINT;                       //  Number of the parameter (correspondence between number andparameter is specified in the table above)
                Value           :   REAL;                       //  New value of the specified parameter
                ExecutionMode   :   AXOpen.Components.Abstractions.Drives.eAxoExecutionMode;          //  Defines the chronological sequence of the method.
            END_VAR
            VAR_OUTPUT
                Done            :   BOOL;                       //  Parameter successfully written
                Busy            :   BOOL;                       //  The method is not finished and new output values are to be expected.
                Error           :   BOOL;                       //  Signals that an error has occurred within the method
                ErrorID         :   DINT;                       //  Error identification
            END_VAR

            _AxoWriteRealParameter_ParameterNumber  :=  ParameterNumber;
            _AxoWriteRealParameter_Value            :=  Value;
            _AxoWriteRealParameter_ExecutionMode    :=  ExecutionMode;

            Done                    :=  AxoWriteRealParameter_Done;
            Busy                    :=  AxoWriteRealParameter_Busy;
            Error                   :=  AxoWriteRealParameter_Error;
            ErrorID                 :=  AxoWriteRealParameter_ErrorID;

            AxoWriteRealParameter   :=  AxoWriteRealParameter_Task.Invoke(THIS);
        END_METHOD

        ///<summary>
        /// This method modifies the value of a vendor specific parameter of type BOOL.
        ///<summary>
        METHOD PUBLIC AxoWriteBoolParameter    : IAxoTaskState
            VAR_INPUT
                ParameterNumber :   DINT;                       //  Number of the parameter (correspondence between number andparameter is specified in the table above)
                Value           :   BOOL;                       //  New value of the specified parameter
                ExecutionMode   :   AXOpen.Components.Abstractions.Drives.eAxoExecutionMode;          //  Defines the chronological sequence of the method.
            END_VAR
            VAR_OUTPUT
                Done            :   BOOL;                       //  Parameter successfully written
                Busy            :   BOOL;                       //  The method is not finished and new output values are to be expected.
                Error           :   BOOL;                       //  Signals that an error has occurred within the method
                ErrorID         :   DINT;                       //  Error identification
            END_VAR

            _AxoWriteBoolParameter_ParameterNumber  :=  ParameterNumber;
            _AxoWriteBoolParameter_Value            :=  Value;
            _AxoWriteBoolParameter_ExecutionMode    :=  ExecutionMode;

            Done                    :=  AxoWriteBoolParameter_Done;
            Busy                    :=  AxoWriteBoolParameter_Busy;
            Error                   :=  AxoWriteBoolParameter_Error;
            ErrorID                 :=  AxoWriteBoolParameter_ErrorID;

            AxoWriteBoolParameter   :=  AxoWriteBoolParameter_Task.Invoke(THIS);
        END_METHOD

        ///<summary>
        /// This method gives access to the value of the input, referenced by the datatype MC_INPUT_REF.
        /// It provides the value of the referenced input (BOOL).
        ///<summary>
        METHOD PUBLIC AxoReadDigitalInput  : IAxoToggleTask
            VAR_INPUT
                Enable          :   BOOL;                       //  Get the value of the selected input signal continuously while enabled
                InputNumber     :   INT;                        //  Selects the input. Can be part of MC_INPUT_REF, if only one single input is referenced.
            END_VAR
            VAR_OUTPUT
                Valid           :   BOOL;                       //  A valid output is available at the method
                Busy            :   BOOL;                       //  The method is not finished and new output values are to be expected
                Error           :   BOOL;                       //  Signals that an error has occurred within the method
                ErrorID         :   DINT;                       //  Error identification
                Value           :   BOOL;                       //  The value of the selected input signal
            END_VAR

            IF Enable THEN
                _AxoReadDigitalInput_InputNumber   :=  InputNumber;

                AxoReadDigitalInput_Task.SwitchOn();
            ELSE
                AxoReadDigitalInput_Task.SwitchOff();
                // THIS.MC_ReadDigitalInput(AxisRef, FALSE);
            END_IF;

            Valid               :=  AxoReadDigitalInput_Valid;
            Busy                :=  AxoReadDigitalInput_Busy;
            Error               :=  AxoReadDigitalInput_Error;
            ErrorID             :=  AxoReadDigitalInput_ErrorID;
            Value               :=  AxoReadDigitalInput_Value;

            AxoReadDigitalInput := AxoReadDigitalInput_Task;
        END_METHOD

        ///<summary>
        /// This method provides access to the value of a digital output, referenced by the datatype MC_OUTPUT_REF.
        /// It provides the value of the referenced output (BOOL).
        ///<summary>
        METHOD PUBLIC AxoReadDigitalOutput : IAxoToggleTask
            VAR_INPUT
                Enable          :   BOOL;                       //  Get the value of the selected output signal continuously while enabled
                OutputNumber    :   INT;                        //  Selects the output. Can be part of MC_OUTPUT_REF, if only one single output is referenced.
            END_VAR
            VAR_OUTPUT
                Valid           :   BOOL;                       //  A valid output is available at the method
                Busy            :   BOOL;                       //  The method is not finished and new output values are to be expected
                Error           :   BOOL;                       //  Signals that an error has occurred within the method
                ErrorID         :   DINT;                       //  Error identification
                Value           :   BOOL;                       //  The value of the selected output signal
            END_VAR

            IF Enable THEN
                _AxoReadDigitalOutput_OutputNumber   :=  OutputNumber;
                AxoReadDigitalOutput_Task.SwitchOn();
            ELSE
                AxoReadDigitalOutput_Task.SwitchOff();
                // THIS.MC_ReadDigitalOutput(AxisRef, FALSE);
            END_IF;

            Valid   := AxoReadDigitalOutput_Valid;
            Busy    :=  AxoReadDigitalOutput_Busy;
            Error   :=  AxoReadDigitalOutput_Error;
            ErrorID :=  AxoReadDigitalOutput_ErrorID;
            Value   := AxoReadDigitalOutput_Value;

            AxoReadDigitalOutput  := AxoReadDigitalOutput_Task;
        END_METHOD

        ///<summary>
        /// This method writes a value to the output referenced by the argument ‘Output’ once (with rising edge of Execute)
        ///<summary>
        METHOD PUBLIC AxoWriteDigitalOutput    : IAxoTaskState
            VAR_INPUT
                OutputNumber    :   INT;                        //  Selects the output. Can be part of MC_OUTPUT_REF, if only one single output is referenced.
                Value           :   BOOL;                       //  The value of the selected output signal
                ExecutionMode   :   AXOpen.Components.Abstractions.Drives.eAxoExecutionMode;          //  Defines the chronological sequence of the method.
            END_VAR
            VAR_OUTPUT
                Done            :   BOOL;                       //  Writing of the output signal value is done
                Busy            :   BOOL;                       //  The method is not finished and new output values are to be expected.
                Error           :   BOOL;                       //  Signals that an error has occurred within the method
                ErrorID         :   DINT;                       //  Error identification
            END_VAR

            _AxoWriteDigitalOutput_OutputNumber     :=  OutputNumber;
            _AxoWriteDigitalOutput_Value            :=  Value;
            _AxoWriteDigitalOutput_ExecutionMode    :=  ExecutionMode;

            Done        :=  AxoWriteDigitalOutput_Done;
            Busy        :=  AxoWriteDigitalOutput_Busy;
            Error       :=  AxoWriteDigitalOutput_Error;
            ErrorID     :=  AxoWriteDigitalOutput_ErrorID;

            AxoWriteDigitalOutput   := AxoWriteDigitalOutput_Task.Invoke(THIS);
        END_METHOD

        ///<summary>
        /// This method returns the actual position.
        ///<summary>
        METHOD PUBLIC AxoReadActualPosition : IAxoToggleTask
            VAR_INPUT
                Enable          :   BOOL;                       //  Get the value of the parameter continuously while enabled
            END_VAR
            VAR_OUTPUT
                Valid           :   BOOL;                       //  A valid output is available at the method
                Busy            :   BOOL;                       //  The method is not finished and new output values are to be expected
                Error           :   BOOL;                       //  Signals that an error has occurred within the method
                ErrorID         :   DINT;                       //  Error identification
                Position        :   LREAL;                      //  New absolute position (in axis’ unit [u])
            END_VAR
